TYPE WAAGE_VAR :
STRUCT
	(*für Verknüpfung mit der Klemme EL6002*)

//in Daten
    EL6002_in AT %I*: EL6inData22B;				// wird mit COM TxPDO Status verknüpft und mit COM TxPDO Data Inxx multiverknüpft
  					
//out Daten
	EL6002_out AT %Q*: EL6outData22B;			// wird mit COM RxPDO Ctrl verknüpft und mit COM RxPDO Data Outxx multiverknüpft

	Masse				: REAL;					// angegeben in [gr]		
	bStabilerWert      	: BOOL;					// wird TRUE falls der ausgegebene Wert stabil ist
	Nummer				: INT;					// 1 bis 4 sind verteilt
	xPosition			: REAL;					// [mm]; relativ zum 2D-Mittelpunkt des Wärmeübertragers im VD
	yPosition			: REAL;					// [mm]; relativ zum 2D-Mittelpunkt des Wärmeübertragers im VD
	k_ist 				: REAL := 0.5;
END_STRUCT
END_TYPE

(* stored: Version 1.1.0.1, ProductVersion 3.1.4019.2
   DUT WAAGE_VAR: Id {02166590-eac0-43fe-9e94-88f3d5299a78} *)
